# EPICS StreamDevice protocol: data/Lakeshore340.proto
Terminator = LF;

getTempA {
  out "KRDG? 0";
  in "%e";
}

setTempA {
  out "SETP 1,%f";
}

getSetTempA {
  out "SETP? 1";
  in "%e";
}

getTempB {
  out "KRDG? 1";
  in "%e";
}

getTempC {
  out "KRDG? 2";
  in "%e";
}

getTempD {
  out "KRDG? 3";
  in "%e";
}

getRdgA {
  out "SRDG? 0";
  in "%e";
}

getRdgB {
  out "SRDG? 1";
  in "%e";
}

getRdgC {
  out "SRDG? 2";
  in "%e";
}

getRdgD {
  out "SRDG? 3";
  in "%e";
}

setP {
  out "PID 1,%f,%(\$1I)f,%(\$1D)d";
  out "PID? 1";
  in "%(\$1P)f,%(\$1I)f,%(\$1D)d"
}

getP {
  out "PID? 1";
  in "%f,%*f,%*d";
}

setI {
  out "PID 1,%(\$1P)f,%f,%(\$1D)d";
  out "PID? 1";
  in "%(\$1P)f,%(\$1I)f,%(\$1D)d"
}

getI {
  out "PID? 1";
  in "%*f,%f,%*d";
}

setD {
  out "PID 1,%(\$1P)f,%(\$1I)f,%d";
  out "PID? 1";
  in "%(\$1P)f,%(\$1I)f,%(\$1D)d"
}

getD {
  out "PID? 1";
  in "%*f,%*f,%d";
}
